# B&R Automation Studio project MotionTestBenchMaster (part 49)

```iecst
                               VAR_DOS_SEQ.Device.LTJ203.ALR_HighLimitEn := TRUE;                                      (* STEP: 9 Hema Tank Level*)
                               VAR_DOS_SEQ.Device.LTJ203.ALR_HighLimitSP := HMI_PAM_3._607;
                               VAR_DOS_SEQ.Device.LTJ203.ALR_LowLimitEn := FALSE;
                               VAR_DOS_SEQ.Device.LTJ203.ALR_LowLimitSP := 0;
                               VAR_DOS_SEQ.Device.LTJ203.SP := 55;
                               VAR_DOS_SEQ.Device.LTJ203.CMP := 3;
                               VAR_DOS_SEQ.Device.LTJ203.MinDev := 0;
                               VAR_DOS_SEQ.Device.LTJ203.MaxDev := 0;

                               VAR_DOS_SEQ.Device.TTJ203.ALR_HighLimitEn := TRUE;                                      (* STEP: 9 Hema Tank Temperature*)
                               VAR_DOS_SEQ.Device.TTJ203.ALR_HighLimitSP := HMI_PAM_3._604;
                               VAR_DOS_SEQ.Device.TTJ203.ALR_LowLimitEn := FALSE;
                               VAR_DOS_SEQ.Device.TTJ203.ALR_LowLimitSP := 0;
                               VAR_DOS_SEQ.Device.TTJ203.SP := 40;
                               VAR_DOS_SEQ.Device.TTJ203.CMP := 2;
                               VAR_DOS_SEQ.Device.TTJ203.MinDev := 0;
                               VAR_DOS_SEQ.Device.TTJ203.MaxDev := 0;

                               VAR_DOS_SEQ.Device.LSJ200.ALR := FALSE;                                                 (* STEP: 9 *)
                               VAR_DOS_SEQ.Device.LSJ200.WAIT_OFF := FALSE;
                               VAR_DOS_SEQ.Device.LSJ200.WAIT_ON := FALSE;

                               VAR_DOS_SEQ.Device.LSJ201.ALR := FALSE;                                                 (* STEP: 9 *)
                               VAR_DOS_SEQ.Device.LSJ201.WAIT_OFF := FALSE;
                               VAR_DOS_SEQ.Device.LSJ201.WAIT_ON := FALSE;

                               VAR_DOS_SEQ.Device.LSJ202.ALR := FALSE;                                                 (* STEP: 9 *)
                               VAR_DOS_SEQ.Device.LSJ202.WAIT_OFF := FALSE;
                               VAR_DOS_SEQ.Device.LSJ202.WAIT_ON := FALSE;

                               VAR_DOS_SEQ.Device.FSJ201.ALR := FALSE;                                                 (* STEP: 9 *)
                               VAR_DOS_SEQ.Device.FSJ201.WAIT_OFF := FALSE;
                               VAR_DOS_SEQ.Device.FSJ201.WAIT_ON := FALSE;

                               VAR_DOS_SEQ.Device.FSJ202.ALR := FALSE;                                                 (* STEP: 9 *)
                               VAR_DOS_SEQ.Device.FSJ202.WAIT_OFF := FALSE;
                               VAR_DOS_SEQ.Device.FSJ202.WAIT_ON := FALSE;

                               VAR_DOS_SEQ.Mem.PBAbortEnable := TRUE;                                                  (* STEP: 9 PB Abort Sequence Enable*)
                               VAR_DOS_SEQ.Mem.PBStopEnable := TRUE;                                                   (* STEP: 9 PB Stop Sequence Enable*)
                               VAR_DOS_SEQ.Mem.PBStartEnable := FALSE;                                                 (* STEP: 9 PB Start Sequence Enable*)
                               VAR_DOS_SEQ.Mem.ContainersStop := TRUE;                                                 (* STEP: 9 *)
                               VAR_DOS_SEQ.Mem.MachineStart := FALSE;                                                  (* STEP: 9 *)
                               VAR_DOS_SEQ.Mem.MachineStop := FALSE;                                                   (* STEP: 9 *)
                               VAR_DOS_SEQ.Mem.DummyBottles := FALSE;                                                  (* STEP: 9 Dummy Bottle Install*)
                               VAR_DOS_SEQ.Mem.PositioningRequest := FALSE;                                            (* STEP: 9 Request of Cam Positioning at height SP of Sequncer*)
                               VAR_DOS_SEQ.Mem.COP_Cycle := FALSE;                                                     (* STEP: 9 COP Cycle Check Requested*)
                               VAR_DOS_SEQ.Mem.LapsCounter := FALSE;                                                   (* STEP: 9 *)
                               VAR_DOS_SEQ.Mem.ValveOpening := TRUE;                                                   (* STEP: 9 *)
                               VAR_DOS_SEQ.Mem.CopAfterCipRequest := FALSE;                                            (* STEP: 9 Request Of Cop After Cip*)

                               VAR_DOS_SEQ.ITC.CIP_CleaningRequest := FALSE;                                           (* STEP: 9 To CIP -> Request of Solution Sending*)
                               VAR_DOS_SEQ.ITC.CIP_Alarm := FALSE;                                                     (* STEP: 9 To CIP -> Critical Alarm Present*)
                               VAR_DOS_SEQ.ITC.CIP_RinseEnded := FALSE;                                                (* STEP: 9 To CIP -> Rinse Finished*)
                               VAR_DOS_SEQ.ITC.CIP_ChangeEnded := FALSE;                                               (* STEP: 9 To CIP -> Change Finished*)
                               VAR_DOS_SEQ.ITC.CIP_DrainRunning := FALSE;                                              (* STEP: 9 To CIP -> Drain Cycle Running*)
                               VAR_DOS_SEQ.ITC.CIP_RinseRunning := FALSE;                                              (* STEP: 9 To CIP -> Rinse Cycle Running*)
                               VAR_DOS_SEQ.ITC.CIP_CleaningRunning := FALSE;                                           (* STEP: 9 To CIP -> Cleaning Cycle Running*)
                               VAR_DOS_SEQ.ITC.CIP_DrainEnded := FALSE;                                                (* STEP: 9 To CIP -> Drain Finished*)
                               VAR_DOS_SEQ.ITC.CIP_FloodingEnded := FALSE;                                             (* STEP: 9 To CIP -> Flooding Finished*)
                               VAR_DOS_SEQ.ITC.CIP_FlipEnable := FALSE;                                                (* STEP: 9 *)
                               VAR_DOS_SEQ.ITC.CIP_CycleEnded := FALSE;                                                (* STEP: 9 *)

                               VAR_DOS_SEQ.ITC.PROD_ReadyForHeating := TRUE;                                           (* STEP: 9 To PASTO -> Filler Ready for Production (Heating)*)
                               VAR_DOS_SEQ.ITC.PROD_DoserInTemperature := FALSE;                                       (* STEP: 9 To PASTO -> Filler Temperature OK (After Heating)*)
                               VAR_DOS_SEQ.ITC.PROD_ProductRequest := FALSE;                                           (* STEP: 9 To PASTO -> Product Request*)
                               VAR_DOS_SEQ.ITC.PROD_DoserOnFillingMode := FALSE;                                       (* STEP: 9 To PASTO -> Product Consumend -Filling Valve Opening*)
                               VAR_DOS_SEQ.ITC.PROD_EndProductionCompleted := FALSE;                                   (* STEP: 9 To PASTO -> End Production Done*)
                               VAR_DOS_SEQ.ITC.PROD_ProductRecoveryEnd := FALSE;                                       (* STEP: 9 To PASTO -> Product Recovery End*)
                               VAR_DOS_SEQ.ITC.PROD_WaterRequestAfterProd := FALSE;                                    (* STEP: 9 To PASTO -> Water Request For Filler Rinse Afetr Production*)

                       10..14: (* Spare Steps *)

                       15: (* START-UP PRODUCTION -Machine Pipes Drainages *)

                               VAR_DOS_SEQ.Device.PPJ201_PID.PID_Enable := FALSE;                                      (* STEP: 15 Doser Recovery Pump*)
                               VAR_DOS_SEQ.Device.PPJ201_PID.PID_Mode := FALSE;
                               VAR_DOS_SEQ.Device.PPJ201_PID.Auto_SP_Value := 0;
                               VAR_DOS_SEQ.Device.PPJ201_PID.FIX_Value := 0;

                               VAR_DOS_SEQ.Device.PPJ202_PID.PID_Enable := FALSE;                                      (* STEP: 15 Doser Recovery Pump*)
                               VAR_DOS_SEQ.Device.PPJ202_PID.PID_Mode := FALSE;
                               VAR_DOS_SEQ.Device.PPJ202_PID.Auto_SP_Value := 0;
                               VAR_DOS_SEQ.Device.PPJ202_PID.FIX_Value := 0;

                               VAR_DOS_SEQ.Device.PPJ203_PID.PID_Enable := FALSE;                                      (* STEP: 15 Diaphragm Pump for Recovery pulp*)
                               VAR_DOS_SEQ.Device.PPJ203_PID.PID_Mode := FALSE;
                               VAR_DOS_SEQ.Device.PPJ203_PID.Auto_SP_Value := 0;
                               VAR_DOS_SEQ.Device.PPJ203_PID.FIX_Value := 0;

                               VAR_DOS_SEQ.Device.MMJ201_PID.PID_Enable := FALSE;                                      (* STEP: 15 Shaker Motor*)
                               VAR_DOS_SEQ.Device.MMJ201_PID.PID_Mode := FALSE;
                               VAR_DOS_SEQ.Device.MMJ201_PID.Auto_SP_Value := 0;
                               VAR_DOS_SEQ.Device.MMJ201_PID.FIX_Value := 0;

                               VAR_DOS_SEQ.Device.RVJ201_PID.PID_Enable := FALSE;                                      (* STEP: 15 *)
                               VAR_DOS_SEQ.Device.RVJ201_PID.PID_Mode := FALSE;
                               VAR_DOS_SEQ.Device.RVJ201_PID.Auto_SP_Value := 0;
                               VAR_DOS_SEQ.Device.RVJ201_PID.FIX_Value := 0;

                               VAR_DOS_SEQ.Device.AVJ201.AutoCnd := FALSE;                                             (* STEP: 15 Inlet Valve*)
                               VAR_DOS_SEQ.Device.AVJ201.EnableCnd := FALSE;
                               VAR_DOS_SEQ.Device.AVJ210.AutoCnd := FALSE;                                             (* STEP: 15 Washing Duct Valve*)
                               VAR_DOS_SEQ.Device.AVJ210.EnableCnd := FALSE;
                               VAR_DOS_SEQ.Device.AVJ211.AutoCnd := FALSE;                                             (* STEP: 15 Sprayball Valve*)
                               VAR_DOS_SEQ.Device.AVJ211.EnableCnd := FALSE;
                               VAR_DOS_SEQ.Device.AVJ212.AutoCnd := FALSE;                                             (* STEP: 15 *)
                               VAR_DOS_SEQ.Device.AVJ212.EnableCnd := FALSE;
                               VAR_DOS_SEQ.Device.AVJ215.AutoCnd := TRUE;                                              (* STEP: 15 Atmospheric drain valve*)
                               VAR_DOS_SEQ.Device.AVJ215.EnableCnd := FALSE;
                               VAR_DOS_SEQ.Device.AVJ216.AutoCnd := FALSE;                                             (* STEP: 15 Recirculation Valve*)
                               VAR_DOS_SEQ.Device.AVJ216.EnableCnd := FALSE;
                               VAR_DOS_SEQ.Device.AVJ217.AutoCnd := TRUE;                                              (* STEP: 15 Tank Hema Drain Valve*)
                               VAR_DOS_SEQ.Device.AVJ217.EnableCnd := FALSE;
                               VAR_DOS_SEQ.Device.AVJ218.AutoCnd := FALSE;                                             (* STEP: 15 Recirculation Valve*)
                               VAR_DOS_SEQ.Device.AVJ218.EnableCnd := FALSE;
                               VAR_DOS_SEQ.Device.AVJ221.AutoCnd := FALSE;                                             (* STEP: 15 Inlet Loop Valve*)
                               VAR_DOS_SEQ.Device.AVJ221.EnableCnd := FALSE;
                               VAR_DOS_SEQ.Device.AVJ230.AutoCnd := FALSE;                                             (* STEP: 15 *)
                               VAR_DOS_SEQ.Device.AVJ230.EnableCnd := FALSE;
                               VAR_DOS_SEQ.Device.AVJ231.AutoCnd := FALSE;                                             (* STEP: 15 *)
                               VAR_DOS_SEQ.Device.AVJ231.EnableCnd := FALSE;
                               VAR_DOS_SEQ.Device.AVJ232.AutoCnd := TRUE;                                              (* STEP: 15 *)
                               VAR_DOS_SEQ.Device.AVJ232.EnableCnd := FALSE;
                               VAR_DOS_SEQ.Device.AVJ233.AutoCnd := FALSE;                                             (* STEP: 15 *)
                               VAR_DOS_SEQ.Device.AVJ233.EnableCnd := FALSE;
                               VAR_DOS_SEQ.Device.AVJ234.AutoCnd := FALSE;                                             (* STEP: 15 *)
                               VAR_DOS_SEQ.Device.AVJ234.EnableCnd := FALSE;
                               VAR_DOS_SEQ.Device.AVJ235.AutoCnd := TRUE;                                              (* STEP: 15 *)
                               VAR_DOS_SEQ.Device.AVJ235.EnableCnd := FALSE;

                               VAR_DOS_SEQ.Device.LTJ203.ALR_HighLimitEn := FALSE;                                     (* STEP: 15 Hema Tank Level*)
                               VAR_DOS_SEQ.Device.LTJ203.ALR_HighLimitSP := 0;
                               VAR_DOS_SEQ.Device.LTJ203.ALR_LowLimitEn := FALSE;
                               VAR_DOS_SEQ.Device.LTJ203.ALR_LowLimitSP := 0;
                               VAR_DOS_SEQ.Device.LTJ203.SP := 5;
                               VAR_DOS_SEQ.Device.LTJ203.CMP := 1;
                               VAR_DOS_SEQ.Device.LTJ203.MinDev := 1;
                               VAR_DOS_SEQ.Device.LTJ203.MaxDev := 1;

                               VAR_DOS_SEQ.Device.TTJ203.ALR_HighLimitEn := FALSE;                                     (* STEP: 15 Hema Tank Temperature*)
                               VAR_DOS_SEQ.Device.TTJ203.ALR_HighLimitSP := 0;
                               VAR_DOS_SEQ.Device.TTJ203.ALR_LowLimitEn := FALSE;
                               VAR_DOS_SEQ.Device.TTJ203.ALR_LowLimitSP := 0;
                               VAR_DOS_SEQ.Device.TTJ203.SP := 0;
                               VAR_DOS_SEQ.Device.TTJ203.CMP := 0;
                               VAR_DOS_SEQ.Device.TTJ203.MinDev := 0;
                               VAR_DOS_SEQ.Device.TTJ203.MaxDev := 0;

                               VAR_DOS_SEQ.Device.LSJ200.ALR := FALSE;                                                 (* STEP: 15 *)
                               VAR_DOS_SEQ.Device.LSJ200.WAIT_OFF := FALSE;
                               VAR_DOS_SEQ.Device.LSJ200.WAIT_ON := FALSE;

                               VAR_DOS_SEQ.Device.LSJ201.ALR := FALSE;                                                 (* STEP: 15 *)
                               VAR_DOS_SEQ.Device.LSJ201.WAIT_OFF := FALSE;
                               VAR_DOS_SEQ.Device.LSJ201.WAIT_ON := FALSE;

                               VAR_DOS_SEQ.Device.LSJ202.ALR := FALSE;                                                 (* STEP: 15 *)
                               VAR_DOS_SEQ.Device.LSJ202.WAIT_OFF := FALSE;
                               VAR_DOS_SEQ.Device.LSJ202.WAIT_ON := FALSE;

                               VAR_DOS_SEQ.Device.FSJ201.ALR := FALSE;                                                 (* STEP: 15 *)
                               VAR_DOS_SEQ.Device.FSJ201.WAIT_OFF := FALSE;
                               VAR_DOS_SEQ.Device.FSJ201.WAIT_ON := FALSE;

                               VAR_DOS_SEQ.Device.FSJ202.ALR := FALSE;                                                 (* STEP: 15 *)
                               VAR_DOS_SEQ.Device.FSJ202.WAIT_OFF := FALSE;
                               VAR_DOS_SEQ.Device.FSJ202.WAIT_ON := FALSE;

                               VAR_DOS_SEQ.Mem.PBAbortEnable := TRUE;                                                  (* STEP: 15 PB Abort Sequence Enable*)
                               VAR_DOS_SEQ.Mem.PBStopEnable := TRUE;                                                   (* STEP: 15 PB Stop Sequence Enable*)
                               VAR_DOS_SEQ.Mem.PBStartEnable := FALSE;                                                 (* STEP: 15 PB Start Sequence Enable*)
                               VAR_DOS_SEQ.Mem.ContainersStop := TRUE;                                                (* STEP: 15 *)
                               VAR_DOS_SEQ.Mem.MachineStart := TRUE;                                                   (* STEP: 15 *)
                               VAR_DOS_SEQ.Mem.MachineStop := FALSE;                                                   (* STEP: 15 *)
                               VAR_DOS_SEQ.Mem.DummyBottles := FALSE;                                                  (* STEP: 15 Dummy Bottle Install*)
                               VAR_DOS_SEQ.Mem.PositioningRequest := FALSE;                                            (* STEP: 15 Request of Cam Positioning at height SP of Sequncer*)
                               VAR_DOS_SEQ.Mem.COP_Cycle := FALSE;                                                     (* STEP: 15 COP Cycle Check Requested*)
                               VAR_DOS_SEQ.Mem.LapsCounter := FALSE;                                                   (* STEP: 15 *)
                               VAR_DOS_SEQ.Mem.ValveOpening := FALSE;                                                  (* STEP: 15 *)
                               VAR_DOS_SEQ.Mem.CopAfterCipRequest := FALSE;                                            (* STEP: 15 Request Of Cop After Cip*)

                               VAR_DOS_SEQ.ITC.CIP_CleaningRequest := FALSE;                                           (* STEP: 15 To CIP -> Request of Solution Sending*)
                               VAR_DOS_SEQ.ITC.CIP_Alarm := FALSE;                                                     (* STEP: 15 To CIP -> Critical Alarm Present*)
                               VAR_DOS_SEQ.ITC.CIP_RinseEnded := FALSE;                                                (* STEP: 15 To CIP -> Rinse Finished*)
                               VAR_DOS_SEQ.ITC.CIP_ChangeEnded := FALSE;                                               (* STEP: 15 To CIP -> Change Finished*)
                               VAR_DOS_SEQ.ITC.CIP_DrainRunning := FALSE;                                              (* STEP: 15 To CIP -> Drain Cycle Running*)
                               VAR_DOS_SEQ.ITC.CIP_RinseRunning := FALSE;                                              (* STEP: 15 To CIP -> Rinse Cycle Running*)
                               VAR_DOS_SEQ.ITC.CIP_CleaningRunning := FALSE;                                           (* STEP: 15 To CIP -> Cleaning Cycle Running*)
                               VAR_DOS_SEQ.ITC.CIP_DrainEnded := FALSE;                                                (* STEP: 15 To CIP -> Drain Finished*)
                               VAR_DOS_SEQ.ITC.CIP_FloodingEnded := FALSE;                                             (* STEP: 15 To CIP -> Flooding Finished*)
                               VAR_DOS_SEQ.ITC.CIP_FlipEnable := FALSE;                                                (* STEP: 15 *)
                               VAR_DOS_SEQ.ITC.CIP_CycleEnded := FALSE;                                                (* STEP: 15 *)

                               VAR_DOS_SEQ.ITC.PROD_ReadyForHeating := FALSE;                                          (* STEP: 15 To PASTO -> Filler Ready for Production (Heating)*)
                               VAR_DOS_SEQ.ITC.PROD_DoserInTemperature := TRUE;                                        (* STEP: 15 To PASTO -> Filler Temperature OK (After Heating)*)
                               VAR_DOS_SEQ.ITC.PROD_ProductRequest := FALSE;                                           (* STEP: 15 To PASTO -> Product Request*)
                               VAR_DOS_SEQ.ITC.PROD_DoserOnFillingMode := FALSE;                                       (* STEP: 15 To PASTO -> Product Consumend -Filling Valve Opening*)
                               VAR_DOS_SEQ.ITC.PROD_EndProductionCompleted := FALSE;                                   (* STEP: 15 To PASTO -> End Production Done*)
                               VAR_DOS_SEQ.ITC.PROD_ProductRecoveryEnd := FALSE;                                       (* STEP: 15 To PASTO -> Product Recovery End*)
                               VAR_DOS_SEQ.ITC.PROD_WaterRequestAfterProd := FALSE;                                    (* STEP: 15 To PASTO -> Water Request For Filler Rinse Afetr Production*)

                       16: (* Spare Steps *)

                       17: (* START-UP PRODUCTION -Machine Draining End *)

                               VAR_DOS_SEQ.Device.PPJ201_PID.PID_Enable := FALSE;                                      (* STEP: 17 Doser Recovery Pump*)
                               VAR_DOS_SEQ.Device.PPJ201_PID.PID_Mode := FALSE;
                               VAR_DOS_SEQ.Device.PPJ201_PID.Auto_SP_Value := 0;
                               VAR_DOS_SEQ.Device.PPJ201_PID.FIX_Value := 0;

                               VAR_DOS_SEQ.Device.PPJ202_PID.PID_Enable := FALSE;                                      (* STEP: 17 Doser Recovery Pump*)
                               VAR_DOS_SEQ.Device.PPJ202_PID.PID_Mode := FALSE;
                               VAR_DOS_SEQ.Device.PPJ202_PID.Auto_SP_Value := 0;
                               VAR_DOS_SEQ.Device.PPJ202_PID.FIX_Value := 0;

                               VAR_DOS_SEQ.Device.PPJ203_PID.PID_Enable := FALSE;                                      (* STEP: 17 Diaphragm Pump for Recovery pulp*)
                               VAR_DOS_SEQ.Device.PPJ203_PID.PID_Mode := FALSE;
                               VAR_DOS_SEQ.Device.PPJ203_PID.Auto_SP_Value := 0;
                               VAR_DOS_SEQ.Device.PPJ203_PID.FIX_Value := 0;

                               VAR_DOS_SEQ.Device.MMJ201_PID.PID_Enable := FALSE;                                      (* STEP: 17 Shaker Motor*)
                               VAR_DOS_SEQ.Device.MMJ201_PID.PID_Mode := FALSE;
                               VAR_DOS_SEQ.Device.MMJ201_PID.Auto_SP_Value := 0;
                               VAR_DOS_SEQ.Device.MMJ201_PID.FIX_Value := 0;

                               VAR_DOS_SEQ.Device.RVJ201_PID.PID_Enable := FALSE;                                      (* STEP: 17 *)
                               VAR_DOS_SEQ.Device.RVJ201_PID.PID_Mode := FALSE;
                               VAR_DOS_SEQ.Device.RVJ201_PID.Auto_SP_Value := 0;
                               VAR_DOS_SEQ.Device.RVJ201_PID.FIX_Value := 0;

                               VAR_DOS_SEQ.Device.AVJ201.AutoCnd := FALSE;                                             (* STEP: 17 Inlet Valve*)
                               VAR_DOS_SEQ.Device.AVJ201.EnableCnd := FALSE;
                               VAR_DOS_SEQ.Device.AVJ210.AutoCnd := FALSE;                                             (* STEP: 17 Washing Duct Valve*)
                               VAR_DOS_SEQ.Device.AVJ210.EnableCnd := FALSE;
                               VAR_DOS_SEQ.Device.AVJ211.AutoCnd := FALSE;                                             (* STEP: 17 Sprayball Valve*)
                               VAR_DOS_SEQ.Device.AVJ211.EnableCnd := FALSE;
                               VAR_DOS_SEQ.Device.AVJ212.AutoCnd := FALSE;                                             (* STEP: 17 *)
                               VAR_DOS_SEQ.Device.AVJ212.EnableCnd := FALSE;
                               VAR_DOS_SEQ.Device.AVJ215.AutoCnd := TRUE;                                              (* STEP: 17 Atmospheric drain valve*)
                               VAR_DOS_SEQ.Device.AVJ215.EnableCnd := FALSE;
                               VAR_DOS_SEQ.Device.AVJ216.AutoCnd := FALSE;                                             (* STEP: 17 Recirculation Valve*)
                               VAR_DOS_SEQ.Device.AVJ216.EnableCnd := FALSE;
                               VAR_DOS_SEQ.Device.AVJ217.AutoCnd := TRUE;                                              (* STEP: 17 Tank Hema Drain Valve*)
                               VAR_DOS_SEQ.Device.AVJ217.EnableCnd := FALSE;
                               VAR_DOS_SEQ.Device.AVJ218.AutoCnd := FALSE;                                             (* STEP: 17 Recirculation Valve*)
                               VAR_DOS_SEQ.Device.AVJ218.EnableCnd := FALSE;
                               VAR_DOS_SEQ.Device.AVJ221.AutoCnd := FALSE;                                             (* STEP: 17 Inlet Loop Valve*)
                               VAR_DOS_SEQ.Device.AVJ221.EnableCnd := FALSE;
                               VAR_DOS_SEQ.Device.AVJ230.AutoCnd := FALSE;                                             (* STEP: 17 *)
                               VAR_DOS_SEQ.Device.AVJ230.EnableCnd := FALSE;
                               VAR_DOS_SEQ.Device.AVJ231.AutoCnd := FALSE;                                             (* STEP: 17 *)
                               VAR_DOS_SEQ.Device.AVJ231.EnableCnd := FALSE;
                               VAR_DOS_SEQ.Device.AVJ232.AutoCnd := TRUE;                                              (* STEP: 17 *)
                               VAR_DOS_SEQ.Device.AVJ232.EnableCnd := FALSE;
                               VAR_DOS_SEQ.Device.AVJ233.AutoCnd := FALSE;                                             (* STEP: 17 *)
                               VAR_DOS_SEQ.Device.AVJ233.EnableCnd := FALSE;
                               VAR_DOS_SEQ.Device.AVJ234.AutoCnd := FALSE;                                             (* STEP: 17 *)
                               VAR_DOS_SEQ.Device.AVJ234.EnableCnd := FALSE;
                               VAR_DOS_SEQ.Device.AVJ235.AutoCnd := TRUE;                                              (* STEP: 17 *)
                               VAR_DOS_SEQ.Device.AVJ235.EnableCnd := FALSE;

                               VAR_DOS_SEQ.Device.LTJ203.ALR_HighLimitEn := FALSE;                                     (* STEP: 17 Hema Tank Level*)
                               VAR_DOS_SEQ.Device.LTJ203.ALR_HighLimitSP := 0;
                               VAR_DOS_SEQ.Device.LTJ203.ALR_LowLimitEn := FALSE;
                               VAR_DOS_SEQ.Device.LTJ203.ALR_LowLimitSP := 0;
                               VAR_DOS_SEQ.Device.LTJ203.SP := 0;
                               VAR_DOS_SEQ.Device.LTJ203.CMP := 0;
                               VAR_DOS_SEQ.Device.LTJ203.MinDev := 0;
                               VAR_DOS_SEQ.Device.LTJ203.MaxDev := 0;

                               VAR_DOS_SEQ.Device.TTJ203.ALR_HighLimitEn := FALSE;                                     (* STEP: 17 Hema Tank Temperature*)
                               VAR_DOS_SEQ.Device.TTJ203.ALR_HighLimitSP := 0;
                               VAR_DOS_SEQ.Device.TTJ203.ALR_LowLimitEn := FALSE;
                               VAR_DOS_SEQ.Device.TTJ203.ALR_LowLimitSP := 0;
                               VAR_DOS_SEQ.Device.TTJ203.SP := 0;
                               VAR_DOS_SEQ.Device.TTJ203.CMP := 0;
                               VAR_DOS_SEQ.Device.TTJ203.MinDev := 0;
                               VAR_DOS_SEQ.Device.TTJ203.MaxDev := 0;

                               VAR_DOS_SEQ.Device.LSJ200.ALR := FALSE;                                                 (* STEP: 17 *)
                               VAR_DOS_SEQ.Device.LSJ200.WAIT_OFF := FALSE;
                               VAR_DOS_SEQ.Device.LSJ200.WAIT_ON := FALSE;

                               VAR_DOS_SEQ.Device.LSJ201.ALR := FALSE;                                                 (* STEP: 17 *)
                               VAR_DOS_SEQ.Device.LSJ201.WAIT_OFF := FALSE;
                               VAR_DOS_SEQ.Device.LSJ201.WAIT_ON := FALSE;

                               VAR_DOS_SEQ.Device.LSJ202.ALR := FALSE;                                                 (* STEP: 17 *)
                               VAR_DOS_SEQ.Device.LSJ202.WAIT_OFF := FALSE;
                               VAR_DOS_SEQ.Device.LSJ202.WAIT_ON := FALSE;

                               VAR_DOS_SEQ.Device.FSJ201.ALR := FALSE;                                                 (* STEP: 17 *)
                               VAR_DOS_SEQ.Device.FSJ201.WAIT_OFF := FALSE;
                               VAR_DOS_SEQ.Device.FSJ201.WAIT_ON := FALSE;

                               VAR_DOS_SEQ.Device.FSJ202.ALR := FALSE;                                                 (* STEP: 17 *)
                               VAR_DOS_SEQ.Device.FSJ202.WAIT_OFF := FALSE;
                               VAR_DOS_SEQ.Device.FSJ202.WAIT_ON := FALSE;

                               VAR_DOS_SEQ.Mem.PBAbortEnable := TRUE;                                                  (* STEP: 17 PB Abort Sequence Enable*)
                               VAR_DOS_SEQ.Mem.PBStopEnable := TRUE;                                                   (* STEP: 17 PB Stop Sequence Enable*)
                               VAR_DOS_SEQ.Mem.PBStartEnable := FALSE;                                                 (* STEP: 17 PB Start Sequence Enable*)
                               VAR_DOS_SEQ.Mem.ContainersStop := TRUE;                                                 (* STEP: 17 *)
                               VAR_DOS_SEQ.Mem.MachineStart := FALSE;                                                  (* STEP: 17 *)
                               VAR_DOS_SEQ.Mem.MachineStop := FALSE;                                                   (* STEP: 17 *)
                               VAR_DOS_SEQ.Mem.DummyBottles := FALSE;                                                  (* STEP: 17 Dummy Bottle Install*)
                               VAR_DOS_SEQ.Mem.PositioningRequest := FALSE;                                            (* STEP: 17 Request of Cam Positioning at height SP of Sequncer*)
                               VAR_DOS_SEQ.Mem.COP_Cycle := FALSE;                                                     (* STEP: 17 COP Cycle Check Requested*)
                               VAR_DOS_SEQ.Mem.LapsCounter := FALSE;                                                   (* STEP: 17 *)
                               VAR_DOS_SEQ.Mem.ValveOpening := FALSE;                                                  (* STEP: 17 *)
                               VAR_DOS_SEQ.Mem.CopAfterCipRequest := FALSE;                                            (* STEP: 17 Request Of Cop After Cip*)

                               VAR_DOS_SEQ.ITC.CIP_CleaningRequest := FALSE;                                           (* STEP: 17 To CIP -> Request of Solution Sending*)
                               VAR_DOS_SEQ.ITC.CIP_Alarm := FALSE;                                                     (* STEP: 17 To CIP -> Critical Alarm Present*)
                               VAR_DOS_SEQ.ITC.CIP_RinseEnded := FALSE;                                                (* STEP: 17 To CIP -> Rinse Finished*)
                               VAR_DOS_SEQ.ITC.CIP_ChangeEnded := FALSE;                                               (* STEP: 17 To CIP -> Change Finished*)
                               VAR_DOS_SEQ.ITC.CIP_DrainRunning := FALSE;                                              (* STEP: 17 To CIP -> Drain Cycle Running*)
                               VAR_DOS_SEQ.ITC.CIP_RinseRunning := FALSE;                                              (* STEP: 17 To CIP -> Rinse Cycle Running*)
                               VAR_DOS_SEQ.ITC.CIP_CleaningRunning := FALSE;                                           (* STEP: 17 To CIP -> Cleaning Cycle Running*)
                               VAR_DOS_SEQ.ITC.CIP_DrainEnded := FALSE;                                                (* STEP: 17 To CIP -> Drain Finished*)
                               VAR_DOS_SEQ.ITC.CIP_FloodingEnded := FALSE;                                             (* STEP: 17 To CIP -> Flooding Finished*)
                               VAR_DOS_SEQ.ITC.CIP_FlipEnable := FALSE;                                                (* STEP: 17 *)
                               VAR_DOS_SEQ.ITC.CIP_CycleEnded := FALSE;                                                (* STEP: 17 *)

                               VAR_DOS_SEQ.ITC.PROD_ReadyForHeating := FALSE;                                          (* STEP: 17 To PASTO -> Filler Ready for Production (Heating)*)
                               VAR_DOS_SEQ.ITC.PROD_DoserInTemperature := FALSE;                                       (* STEP: 17 To PASTO -> Filler Temperature OK (After Heating)*)
                               VAR_DOS_SEQ.ITC.PROD_ProductRequest := FALSE;                                           (* STEP: 17 To PASTO -> Product Request*)
                               VAR_DOS_SEQ.ITC.PROD_DoserOnFillingMode := FALSE;                                       (* STEP: 17 To PASTO -> Product Consumend -Filling Valve Opening*)
                               VAR_DOS_SEQ.ITC.PROD_EndProductionCompleted := FALSE;                                   (* STEP: 17 To PASTO -> End Production Done*)
                               VAR_DOS_SEQ.ITC.PROD_ProductRecoveryEnd := FALSE;                                       (* STEP: 17 To PASTO -> Product Recovery End*)
                               VAR_DOS_SEQ.ITC.PROD_WaterRequestAfterProd := FALSE;                                    (* STEP: 17 To PASTO -> Water Request For Filler Rinse Afetr Production*)

                       18..19: (* Spare Steps *)

                       20: (* START-UP PRODUCTION -Wait "Product Available" From PASTO *)

                               VAR_DOS_SEQ.Device.PPJ201_PID.PID_Enable := FALSE;                                      (* STEP: 20 Doser Recovery Pump*)
                               VAR_DOS_SEQ.Device.PPJ201_PID.PID_Mode := FALSE;
                               VAR_DOS_SEQ.Device.PPJ201_PID.Auto_SP_Value := 0;
                               VAR_DOS_SEQ.Device.PPJ201_PID.FIX_Value := 0;

                               VAR_DOS_SEQ.Device.PPJ202_PID.PID_Enable := FALSE;                                      (* STEP: 20 Doser Recovery Pump*)
                               VAR_DOS_SEQ.Device.PPJ202_PID.PID_Mode := FALSE;
                               VAR_DOS_SEQ.Device.PPJ202_PID.Auto_SP_Value := 0;
                               VAR_DOS_SEQ.Device.PPJ202_PID.FIX_Value := 0;

                               VAR_DOS_SEQ.Device.PPJ203_PID.PID_Enable := FALSE;                                      (* STEP: 20 Diaphragm Pump for Recovery pulp*)
                               VAR_DOS_SEQ.Device.PPJ203_PID.PID_Mode := FALSE;
                               VAR_DOS_SEQ.Device.PPJ203_PID.Auto_SP_Value := 0;
                               VAR_DOS_SEQ.Device.PPJ203_PID.FIX_Value := 0;

                               VAR_DOS_SEQ.Device.MMJ201_PID.PID_Enable := FALSE;                                      (* STEP: 20 Shaker Motor*)
                               VAR_DOS_SEQ.Device.MMJ201_PID.PID_Mode := FALSE;
                               VAR_DOS_SEQ.Device.MMJ201_PID.Auto_SP_Value := 0;
                               VAR_DOS_SEQ.Device.MMJ201_PID.FIX_Value := 0;

                               VAR_DOS_SEQ.Device.RVJ201_PID.PID_Enable := FALSE;                                      (* STEP: 20 *)
                               VAR_DOS_SEQ.Device.RVJ201_PID.PID_Mode := FALSE;
                               VAR_DOS_SEQ.Device.RVJ201_PID.Auto_SP_Value := 0;
                               VAR_DOS_SEQ.Device.RVJ201_PID.FIX_Value := 0;

                               VAR_DOS_SEQ.Device.AVJ201.AutoCnd := FALSE;                                             (* STEP: 20 Inlet Valve*)
                               VAR_DOS_SEQ.Device.AVJ201.EnableCnd := FALSE;
                               VAR_DOS_SEQ.Device.AVJ210.AutoCnd := FALSE;                                             (* STEP: 20 Washing Duct Valve*)
                               VAR_DOS_SEQ.Device.AVJ210.EnableCnd := FALSE;
                               VAR_DOS_SEQ.Device.AVJ211.AutoCnd := FALSE;                                             (* STEP: 20 Sprayball Valve*)
                               VAR_DOS_SEQ.Device.AVJ211.EnableCnd := FALSE;
                               VAR_DOS_SEQ.Device.AVJ212.AutoCnd := FALSE;                                             (* STEP: 20 *)
                               VAR_DOS_SEQ.Device.AVJ212.EnableCnd := FALSE;
                               VAR_DOS_SEQ.Device.AVJ215.AutoCnd := TRUE;                                              (* STEP: 20 Atmospheric drain valve *)
                               VAR_DOS_SEQ.Device.AVJ215.EnableCnd := FALSE;
                               VAR_DOS_SEQ.Device.AVJ216.AutoCnd := FALSE;                                             (* STEP: 20 Recirculation Valve*)
                               VAR_DOS_SEQ.Device.AVJ216.EnableCnd := FALSE;
                               VAR_DOS_SEQ.Device.AVJ217.AutoCnd := FALSE;                                              (* STEP: 20 Tank Hema Drain Valve*)
                               VAR_DOS_SEQ.Device.AVJ217.EnableCnd := FALSE;
                               VAR_DOS_SEQ.Device.AVJ218.AutoCnd := FALSE;                                             (* STEP: 20 Recirculation Valve*)
                               VAR_DOS_SEQ.Device.AVJ218.EnableCnd := FALSE;
                               VAR_DOS_SEQ.Device.AVJ221.AutoCnd := FALSE;                                             (* STEP: 20 Inlet Loop Valve*)
                               VAR_DOS_SEQ.Device.AVJ221.EnableCnd := FALSE;
                               VAR_DOS_SEQ.Device.AVJ230.AutoCnd := FALSE;                                             (* STEP: 20 *)
                               VAR_DOS_SEQ.Device.AVJ230.EnableCnd := FALSE;
                               VAR_DOS_SEQ.Device.AVJ231.AutoCnd := FALSE;                                             (* STEP: 20 *)
                               VAR_DOS_SEQ.Device.AVJ231.EnableCnd := FALSE;
                               VAR_DOS_SEQ.Device.AVJ232.AutoCnd := FALSE;                                             (* STEP: 20 *)
                               VAR_DOS_SEQ.Device.AVJ232.EnableCnd := FALSE;
                               VAR_DOS_SEQ.Device.AVJ233.AutoCnd := FALSE;                                             (* STEP: 20 *)
                               VAR_DOS_SEQ.Device.AVJ233.EnableCnd := FALSE;
                               VAR_DOS_SEQ.Device.AVJ234.AutoCnd := FALSE;                                             (* STEP: 20 *)
                               VAR_DOS_SEQ.Device.AVJ234.EnableCnd := FALSE;
                               VAR_DOS_SEQ.Device.AVJ235.AutoCnd := FALSE;                                             (* STEP: 20 *)
                               VAR_DOS_SEQ.Device.AVJ235.EnableCnd := FALSE;

                               VAR_DOS_SEQ.Device.LTJ203.ALR_HighLimitEn := FALSE;                                     (* STEP: 20 Hema Tank Level*)
                               VAR_DOS_SEQ.Device.LTJ203.ALR_HighLimitSP := 0;
                               VAR_DOS_SEQ.Device.LTJ203.ALR_LowLimitEn := FALSE;
                               VAR_DOS_SEQ.Device.LTJ203.ALR_LowLimitSP := 0;
                               VAR_DOS_SEQ.Device.LTJ203.SP := 0;
                               VAR_DOS_SEQ.Device.LTJ203.CMP := 0;
                               VAR_DOS_SEQ.Device.LTJ203.MinDev := 0;
                               VAR_DOS_SEQ.Device.LTJ203.MaxDev := 0;

                               VAR_DOS_SEQ.Device.TTJ203.ALR_HighLimitEn := FALSE;                                     (* STEP: 20 Hema Tank Temperature*)
                               VAR_DOS_SEQ.Device.TTJ203.ALR_HighLimitSP := 0;
                               VAR_DOS_SEQ.Device.TTJ203.ALR_LowLimitEn := FALSE;
                               VAR_DOS_SEQ.Device.TTJ203.ALR_LowLimitSP := 0;
                               VAR_DOS_SEQ.Device.TTJ203.SP := 0;
                               VAR_DOS_SEQ.Device.TTJ203.CMP := 0;
                               VAR_DOS_SEQ.Device.TTJ203.MinDev := 0;
                               VAR_DOS_SEQ.Device.TTJ203.MaxDev := 0;

                               VAR_DOS_SEQ.Device.LSJ200.ALR := FALSE;                                                 (* STEP: 20 *)
                               VAR_DOS_SEQ.Device.LSJ200.WAIT_OFF := FALSE;
                               VAR_DOS_SEQ.Device.LSJ200.WAIT_ON := FALSE;

                               VAR_DOS_SEQ.Device.LSJ201.ALR := FALSE;                                                 (* STEP: 20 *)
                               VAR_DOS_SEQ.Device.LSJ201.WAIT_OFF := FALSE;
                               VAR_DOS_SEQ.Device.LSJ201.WAIT_ON := FALSE;

                               VAR_DOS_SEQ.Device.LSJ202.ALR := FALSE;                                                 (* STEP: 20 *)
                               VAR_DOS_SEQ.Device.LSJ202.WAIT_OFF := FALSE;
                               VAR_DOS_SEQ.Device.LSJ202.WAIT_ON := FALSE;

                               VAR_DOS_SEQ.Device.FSJ201.ALR := FALSE;                                                 (* STEP: 20 *)
                               VAR_DOS_SEQ.Device.FSJ201.WAIT_OFF := FALSE;
                               VAR_DOS_SEQ.Device.FSJ201.WAIT_ON := FALSE;

                               VAR_DOS_SEQ.Device.FSJ202.ALR := FALSE;                                                 (* STEP: 20 *)
                               VAR_DOS_SEQ.Device.FSJ202.WAIT_OFF := FALSE;
                               VAR_DOS_SEQ.Device.FSJ202.WAIT_ON := FALSE;

                               VAR_DOS_SEQ.Mem.PBAbortEnable := TRUE;                                                  (* STEP: 20 PB Abort Sequence Enable*)
                               VAR_DOS_SEQ.Mem.PBStopEnable := TRUE;                                                   (* STEP: 20 PB Stop Sequence Enable*)
                               VAR_DOS_SEQ.Mem.PBStartEnable := FALSE;                                                 (* STEP: 20 PB Start Sequence Enable*)
                               VAR_DOS_SEQ.Mem.ContainersStop := TRUE;                                                 (* STEP: 20 *)
                               VAR_DOS_SEQ.Mem.MachineStart := FALSE;                                                  (* STEP: 20 *)
                               VAR_DOS_SEQ.Mem.MachineStop := FALSE;                                                   (* STEP: 20 *)
                               VAR_DOS_SEQ.Mem.DummyBottles := FALSE;                                                  (* STEP: 20 Dummy Bottle Install*)
                               VAR_DOS_SEQ.Mem.PositioningRequest := FALSE;                                            (* STEP: 20 Request of Cam Positioning at height SP of Sequncer*)
                               VAR_DOS_SEQ.Mem.COP_Cycle := FALSE;                                                     (* STEP: 20 COP Cycle Check Requested*)
                               VAR_DOS_SEQ.Mem.LapsCounter := FALSE;                                                   (* STEP: 20 *)
                               VAR_DOS_SEQ.Mem.ValveOpening := FALSE;                                                  (* STEP: 20 *)
                               VAR_DOS_SEQ.Mem.CopAfterCipRequest := FALSE;                                            (* STEP: 20 Request Of Cop After Cip*)

                               VAR_DOS_SEQ.ITC.CIP_CleaningRequest := FALSE;                                           (* STEP: 20 To CIP -> Request of Solution Sending*)
                               VAR_DOS_SEQ.ITC.CIP_Alarm := FALSE;                                                     (* STEP: 20 To CIP -> Critical Alarm Present*)
                               VAR_DOS_SEQ.ITC.CIP_RinseEnded := FALSE;                                                (* STEP: 20 To CIP -> Rinse Finished*)
                               VAR_DOS_SEQ.ITC.CIP_ChangeEnded := FALSE;                                               (* STEP: 20 To CIP -> Change Finished*)
                               VAR_DOS_SEQ.ITC.CIP_DrainRunning := FALSE;                                              (* STEP: 20 To CIP -> Drain Cycle Running*)
                               VAR_DOS_SEQ.ITC.CIP_RinseRunning := FALSE;                                              (* STEP: 20 To CIP -> Rinse Cycle Running*)
                               VAR_DOS_SEQ.ITC.CIP_CleaningRunning := FALSE;                                           (* STEP: 20 To CIP -> Cleaning Cycle Running*)
                               VAR_DOS_SEQ.ITC.CIP_DrainEnded := FALSE;                                                (* STEP: 20 To CIP -> Drain Finished*)
                               VAR_DOS_SEQ.ITC.CIP_FloodingEnded := FALSE;                                             (* STEP: 20 To CIP -> Flooding Finished*)
                               VAR_DOS_SEQ.ITC.CIP_FlipEnable := FALSE;                                                (* STEP: 20 *)
                               VAR_DOS_SEQ.ITC.CIP_CycleEnded := FALSE;                                                (* STEP: 20 *)

                               VAR_DOS_SEQ.ITC.PROD_ReadyForHeating := FALSE;                                          (* STEP: 20 To PASTO -> Filler Ready for Production (Heating)*)
                               VAR_DOS_SEQ.ITC.PROD_DoserInTemperature := FALSE;                                       (* STEP: 20 To PASTO -> Filler Temperature OK (After Heating)*)
                               VAR_DOS_SEQ.ITC.PROD_ProductRequest := FALSE;                                           (* STEP: 20 To PASTO -> Product Request*)
                               VAR_DOS_SEQ.ITC.PROD_DoserOnFillingMode := FALSE;                                       (* STEP: 20 To PASTO -> Product Consumend -Filling Valve Opening*)
                               VAR_DOS_SEQ.ITC.PROD_EndProductionCompleted := FALSE;                                   (* STEP: 20 To PASTO -> End Production Done*)
                               VAR_DOS_SEQ.ITC.PROD_ProductRecoveryEnd := FALSE;                                       (* STEP: 20 To PASTO -> Product Recovery End*)
                               VAR_DOS_SEQ.ITC.PROD_WaterRequestAfterProd := FALSE;                                    (* STEP: 20 To PASTO -> Water Request For Filler Rinse Afetr Production*)

                       21: (* Spare Steps *)

                       22: (* START-UP PRODUCTION - Load Product at level *)

                               VAR_DOS_SEQ.Device.PPJ201_PID.PID_Enable := FALSE;                                      (* STEP: 22 Doser Recovery Pump*)
                               VAR_DOS_SEQ.Device.PPJ201_PID.PID_Mode := FALSE;
                               VAR_DOS_SEQ.Device.PPJ201_PID.Auto_SP_Value := 0;
                               VAR_DOS_SEQ.Device.PPJ201_PID.FIX_Value := 0;

                               VAR_DOS_SEQ.Device.PPJ202_PID.PID_Enable := FALSE;                                      (* STEP: 22 Doser Recovery Pump*)
                               VAR_DOS_SEQ.Device.PPJ202_PID.PID_Mode := FALSE;
                               VAR_DOS_SEQ.Device.PPJ202_PID.Auto_SP_Value := 0;
                               VAR_DOS_SEQ.Device.PPJ202_PID.FIX_Value := 0;

                               VAR_DOS_SEQ.Device.PPJ203_PID.PID_Enable := FALSE;                                      (* STEP: 22 Diaphragm Pump for Recovery pulp*)
                               VAR_DOS_SEQ.Device.PPJ203_PID.PID_Mode := FALSE;
                               VAR_DOS_SEQ.Device.PPJ203_PID.Auto_SP_Value := 0;
                               VAR_DOS_SEQ.Device.PPJ203_PID.FIX_Value := 0;

                               VAR_DOS_SEQ.Device.MMJ201_PID.PID_Enable := FALSE;                                      (* STEP: 22 Shaker Motor*)
                               VAR_DOS_SEQ.Device.MMJ201_PID.PID_Mode := FALSE;
                               VAR_DOS_SEQ.Device.MMJ201_PID.Auto_SP_Value := 10;
                               VAR_DOS_SEQ.Device.MMJ201_PID.FIX_Value := 0;

                               VAR_DOS_SEQ.Device.RVJ201_PID.PID_Enable := FALSE;                                      (* STEP: 22 *)
                               VAR_DOS_SEQ.Device.RVJ201_PID.PID_Mode := FALSE;
                               VAR_DOS_SEQ.Device.RVJ201_PID.Auto_SP_Value := 0;
                               VAR_DOS_SEQ.Device.RVJ201_PID.FIX_Value := 0;

                               VAR_DOS_SEQ.Device.AVJ201.AutoCnd := TRUE;                                              (* STEP: 22 Inlet Valve*)
                               VAR_DOS_SEQ.Device.AVJ201.EnableCnd := TRUE;
                               VAR_DOS_SEQ.Device.AVJ210.AutoCnd := FALSE;                                             (* STEP: 22 Washing Duct Valve*)
                               VAR_DOS_SEQ.Device.AVJ210.EnableCnd := FALSE;
                               VAR_DOS_SEQ.Device.AVJ211.AutoCnd := FALSE;                                             (* STEP: 22 Sprayball Valve*)
                               VAR_DOS_SEQ.Device.AVJ211.EnableCnd := FALSE;
                               VAR_DOS_SEQ.Device.AVJ212.AutoCnd := FALSE;                                             (* STEP: 22 *)
                               VAR_DOS_SEQ.Device.AVJ212.EnableCnd := FALSE;
                               VAR_DOS_SEQ.Device.AVJ215.AutoCnd := FALSE;                                             (* STEP: 22 Atmospheric drain valve*)
                               VAR_DOS_SEQ.Device.AVJ215.EnableCnd := FALSE;
                               VAR_DOS_SEQ.Device.AVJ216.AutoCnd := FALSE;                                             (* STEP: 22 Recirculation Valve*)
                               VAR_DOS_SEQ.Device.AVJ216.EnableCnd := FALSE;
                               VAR_DOS_SEQ.Device.AVJ217.AutoCnd := FALSE;                                             (* STEP: 22 Tank Hema Drain Valve*)
                               VAR_DOS_SEQ.Device.AVJ217.EnableCnd := FALSE;
                               VAR_DOS_SEQ.Device.AVJ218.AutoCnd := FALSE;                                             (* STEP: 22 Recirculation Valve*)
                               VAR_DOS_SEQ.Device.AVJ218.EnableCnd := FALSE;
                               VAR_DOS_SEQ.Device.AVJ221.AutoCnd := FALSE;                                             (* STEP: 22 Inlet Loop Valve*)
                               VAR_DOS_SEQ.Device.AVJ221.EnableCnd := FALSE;
                               VAR_DOS_SEQ.Device.AVJ230.AutoCnd := FALSE;                                             (* STEP: 22 *)
                               VAR_DOS_SEQ.Device.AVJ230.EnableCnd := FALSE;
                               VAR_DOS_SEQ.Device.AVJ231.AutoCnd := FALSE;                                             (* STEP: 22 *)
                               VAR_DOS_SEQ.Device.AVJ231.EnableCnd := FALSE;
                               VAR_DOS_SEQ.Device.AVJ232.AutoCnd := FALSE;                                             (* STEP: 22 *)
                               VAR_DOS_SEQ.Device.AVJ232.EnableCnd := FALSE;
                               VAR_DOS_SEQ.Device.AVJ233.AutoCnd := FALSE;                                             (* STEP: 22 *)
                               VAR_DOS_SEQ.Device.AVJ233.EnableCnd := FALSE;
                               VAR_DOS_SEQ.Device.AVJ234.AutoCnd := FALSE;                                             (* STEP: 22 *)
                               VAR_DOS_SEQ.Device.AVJ234.EnableCnd := FALSE;
                               VAR_DOS_SEQ.Device.AVJ235.AutoCnd := FALSE;                                             (* STEP: 22 *)
                               VAR_DOS_SEQ.Device.AVJ235.EnableCnd := FALSE;

                               VAR_DOS_SEQ.Device.LTJ203.ALR_HighLimitEn := TRUE;                                      (* STEP: 22 Hema Tank Level*)
                               VAR_DOS_SEQ.Device.LTJ203.ALR_HighLimitSP := HMI_PAM_3._607;
                               VAR_DOS_SEQ.Device.LTJ203.ALR_LowLimitEn := TRUE;
                               VAR_DOS_SEQ.Device.LTJ203.ALR_LowLimitSP := HMI_PAM_3._606;
                               VAR_DOS_SEQ.Device.LTJ203.SP := HMI_PAM_3._608;
                               VAR_DOS_SEQ.Device.LTJ203.CMP := 2;
                               VAR_DOS_SEQ.Device.LTJ203.MinDev := 0;
                               VAR_DOS_SEQ.Device.LTJ203.MaxDev := 0;

                               VAR_DOS_SEQ.Device.TTJ203.ALR_HighLimitEn := FALSE;                                     (* STEP: 22 Hema Tank Temperature*)
                               VAR_DOS_SEQ.Device.TTJ203.ALR_HighLimitSP := 0;
                               VAR_DOS_SEQ.Device.TTJ203.ALR_LowLimitEn := FALSE;
                               VAR_DOS_SEQ.Device.TTJ203.ALR_LowLimitSP := 0;
                               VAR_DOS_SEQ.Device.TTJ203.SP := HMI_PAM_3._600;
                               VAR_DOS_SEQ.Device.TTJ203.CMP := 0;
                               VAR_DOS_SEQ.Device.TTJ203.MinDev := 0;
                               VAR_DOS_SEQ.Device.TTJ203.MaxDev := 0;

                               VAR_DOS_SEQ.Device.LSJ200.ALR := FALSE;                                                 (* STEP: 22 *)
                               VAR_DOS_SEQ.Device.LSJ200.WAIT_OFF := FALSE;
                               VAR_DOS_SEQ.Device.LSJ200.WAIT_ON := FALSE;

                               VAR_DOS_SEQ.Device.LSJ201.ALR := FALSE;                                                 (* STEP: 22 *)
                               VAR_DOS_SEQ.Device.LSJ201.WAIT_OFF := FALSE;
                               VAR_DOS_SEQ.Device.LSJ201.WAIT_ON := FALSE;

                               VAR_DOS_SEQ.Device.LSJ202.ALR := FALSE;                                                 (* STEP: 22 *)
                               VAR_DOS_SEQ.Device.LSJ202.WAIT_OFF := FALSE;
                               VAR_DOS_SEQ.Device.LSJ202.WAIT_ON := FALSE;

                               VAR_DOS_SEQ.Device.FSJ201.ALR := FALSE;                                                 (* STEP: 22 *)
                               VAR_DOS_SEQ.Device.FSJ201.WAIT_OFF := FALSE;
                               VAR_DOS_SEQ.Device.FSJ201.WAIT_ON := FALSE;

                               VAR_DOS_SEQ.Device.FSJ202.ALR := FALSE;                                                 (* STEP: 22 *)
                               VAR_DOS_SEQ.Device.FSJ202.WAIT_OFF := FALSE;
                               VAR_DOS_SEQ.Device.FSJ202.WAIT_ON := FALSE;

                               VAR_DOS_SEQ.Mem.PBAbortEnable := TRUE;                                                  (* STEP: 22 PB Abort Sequence Enable*)
                               VAR_DOS_SEQ.Mem.PBStopEnable := TRUE;                                                   (* STEP: 22 PB Stop Sequence Enable*)
                               VAR_DOS_SEQ.Mem.PBStartEnable := FALSE;                                                 (* STEP: 22 PB Start Sequence Enable*)
                               VAR_DOS_SEQ.Mem.ContainersStop := TRUE;                                                 (* STEP: 22 *)
                               VAR_DOS_SEQ.Mem.MachineStart := TRUE;                                                   (* STEP: 22 *)
                               VAR_DOS_SEQ.Mem.MachineStop := FALSE;                                                   (* STEP: 22 *)
                               VAR_DOS_SEQ.Mem.DummyBottles := FALSE;                                                  (* STEP: 22 Dummy Bottle Install*)
                               VAR_DOS_SEQ.Mem.PositioningRequest := FALSE;                                            (* STEP: 22 Request of Cam Positioning at height SP of Sequncer*)
                               VAR_DOS_SEQ.Mem.COP_Cycle := FALSE;                                                     (* STEP: 22 COP Cycle Check Requested*)
                               VAR_DOS_SEQ.Mem.LapsCounter := FALSE;                                                   (* STEP: 22 *)
                               VAR_DOS_SEQ.Mem.ValveOpening := FALSE;                                                  (* STEP: 22 *)
                               VAR_DOS_SEQ.Mem.CopAfterCipRequest := FALSE;                                            (* STEP: 22 Request Of Cop After Cip*)

                               VAR_DOS_SEQ.ITC.CIP_CleaningRequest := FALSE;                                           (* STEP: 22 To CIP -> Request of Solution Sending*)
                               VAR_DOS_SEQ.ITC.CIP_Alarm := FALSE;                                                     (* STEP: 22 To CIP -> Critical Alarm Present*)
                               VAR_DOS_SEQ.ITC.CIP_RinseEnded := FALSE;                                                (* STEP: 22 To CIP -> Rinse Finished*)
                               VAR_DOS_SEQ.ITC.CIP_ChangeEnded := FALSE;                                               (* STEP: 22 To CIP -> Change Finished*)
                               VAR_DOS_SEQ.ITC.CIP_DrainRunning := FALSE;                                              (* STEP: 22 To CIP -> Drain Cycle Running*)
                               VAR_DOS_SEQ.ITC.CIP_RinseRunning := FALSE;                                              (* STEP: 22 To CIP -> Rinse Cycle Running*)
                               VAR_DOS_SEQ.ITC.CIP_CleaningRunning := FALSE;                                           (* STEP: 22 To CIP -> Cleaning Cycle Running*)
                               VAR_DOS_SEQ.ITC.CIP_DrainEnded := FALSE;                                                (* STEP: 22 To CIP -> Drain Finished*)
                               VAR_DOS_SEQ.ITC.CIP_FloodingEnded := FALSE;                                             (* STEP: 22 To CIP -> Flooding Finished*)
                               VAR_DOS_SEQ.ITC.CIP_FlipEnable := FALSE;                                                (* STEP: 22 *)
                               VAR_DOS_SEQ.ITC.CIP_CycleEnded := FALSE;                                                (* STEP: 22 *)

                               VAR_DOS_SEQ.ITC.PROD_ReadyForHeating := FALSE;                                          (* STEP: 22 To PASTO -> Filler Ready for Production (Heating)*)
                               VAR_DOS_SEQ.ITC.PROD_DoserInTemperature := FALSE;                                       (* STEP: 22 To PASTO -> Filler Temperature OK (After Heating)*)
                               VAR_DOS_SEQ.ITC.PROD_ProductRequest := TRUE;                                            (* STEP: 22 To PASTO -> Product Request*)
                               VAR_DOS_SEQ.ITC.PROD_DoserOnFillingMode := FALSE;                                       (* STEP: 22 To PASTO -> Product Consumend -Filling Valve Opening*)
                               VAR_DOS_SEQ.ITC.PROD_EndProductionCompleted := FALSE;                                   (* STEP: 22 To PASTO -> End Production Done*)
                               VAR_DOS_SEQ.ITC.PROD_ProductRecoveryEnd := FALSE;                                       (* STEP: 22 To PASTO -> Product Recovery End*)
                               VAR_DOS_SEQ.ITC.PROD_WaterRequestAfterProd := FALSE;                                    (* STEP: 22 To PASTO -> Water Request For Filler Rinse Afetr Production*)

                       23: (* START-UP PRODUCTION -Filling Valve Priming, Filling Valves Opening *)

                               VAR_DOS_SEQ.Device.PPJ201_PID.PID_Enable := FALSE;                                      (* STEP: 23 Doser Recovery Pump*)
                               VAR_DOS_SEQ.Device.PPJ201_PID.PID_Mode := FALSE;
                               VAR_DOS_SEQ.Device.PPJ201_PID.Auto_SP_Value := 0;
                               VAR_DOS_SEQ.Device.PPJ201_PID.FIX_Value := 0;

                               VAR_DOS_SEQ.Device.PPJ202_PID.PID_Enable := FALSE;                                      (* STEP: 23 Doser Recovery Pump*)
                               VAR_DOS_SEQ.Device.PPJ202_PID.PID_Mode := FALSE;
                               VAR_DOS_SEQ.Device.PPJ202_PID.Auto_SP_Value := 0;
                               VAR_DOS_SEQ.Device.PPJ202_PID.FIX_Value := 0;

                               VAR_DOS_SEQ.Device.PPJ203_PID.PID_Enable := FALSE;                                      (* STEP: 23 Diaphragm Pump for Recovery pulp*)
                               VAR_DOS_SEQ.Device.PPJ203_PID.PID_Mode := FALSE;
                               VAR_DOS_SEQ.Device.PPJ203_PID.Auto_SP_Value := 0;
                               VAR_DOS_SEQ.Device.PPJ203_PID.FIX_Value := 0;

                               VAR_DOS_SEQ.Device.MMJ201_PID.PID_Enable := FALSE;                                      (* STEP: 23 Shaker Motor*)
                               VAR_DOS_SEQ.Device.MMJ201_PID.PID_Mode := FALSE;
                               VAR_DOS_SEQ.Device.MMJ201_PID.Auto_SP_Value := 10;
                               VAR_DOS_SEQ.Device.MMJ201_PID.FIX_Value := 0;

                               VAR_DOS_SEQ.Device.RVJ201_PID.PID_Enable := FALSE;                                      (* STEP: 23 *)
                               VAR_DOS_SEQ.Device.RVJ201_PID.PID_Mode := FALSE;
                               VAR_DOS_SEQ.Device.RVJ201_PID.Auto_SP_Value := 0;
                               VAR_DOS_SEQ.Device.RVJ201_PID.FIX_Value := 0;

                               VAR_DOS_SEQ.Device.AVJ201.AutoCnd := TRUE;                                              (* STEP: 23 Inlet Valve*)
                               VAR_DOS_SEQ.Device.AVJ201.EnableCnd := TRUE;
                               VAR_DOS_SEQ.Device.AVJ210.AutoCnd := FALSE;                                             (* STEP: 23 Washing Duct Valve*)
                               VAR_DOS_SEQ.Device.AVJ210.EnableCnd := FALSE;
                               VAR_DOS_SEQ.Device.AVJ211.AutoCnd := FALSE;                                             (* STEP: 23 Sprayball Valve*)
                               VAR_DOS_SEQ.Device.AVJ211.EnableCnd := FALSE;
                               VAR_DOS_SEQ.Device.AVJ212.AutoCnd := FALSE;                                             (* STEP: 23 *)
                               VAR_DOS_SEQ.Device.AVJ212.EnableCnd := FALSE;
                               VAR_DOS_SEQ.Device.AVJ215.AutoCnd := FALSE;                                             (* STEP: 23 Atmospheric drain valve*)
                               VAR_DOS_SEQ.Device.AVJ215.EnableCnd := FALSE;
                               VAR_DOS_SEQ.Device.AVJ216.AutoCnd := FALSE;                                             (* STEP: 23 Recirculation Valve*)
                               VAR_DOS_SEQ.Device.AVJ216.EnableCnd := FALSE;
                               VAR_DOS_SEQ.Device.AVJ217.AutoCnd := FALSE;                                             (* STEP: 23 Tank Hema Drain Valve*)
                               VAR_DOS_SEQ.Device.AVJ217.EnableCnd := FALSE;
                               VAR_DOS_SEQ.Device.AVJ218.AutoCnd := FALSE;                                             (* STEP: 23 Recirculation Valve*)
                               VAR_DOS_SEQ.Device.AVJ218.EnableCnd := FALSE;
                               VAR_DOS_SEQ.Device.AVJ221.AutoCnd := FALSE;                                             (* STEP: 23 Inlet Loop Valve*)
                               VAR_DOS_SEQ.Device.AVJ221.EnableCnd := FALSE;
                               VAR_DOS_SEQ.Device.AVJ230.AutoCnd := FALSE;                                             (* STEP: 23 *)
                               VAR_DOS_SEQ.Device.AVJ230.EnableCnd := FALSE;
                               VAR_DOS_SEQ.Device.AVJ231.AutoCnd := FALSE;                                             (* STEP: 23 *)
                               VAR_DOS_SEQ.Device.AVJ231.EnableCnd := FALSE;
                               VAR_DOS_SEQ.Device.AVJ232.AutoCnd := TRUE;                                              (* STEP: 23 *)
                               VAR_DOS_SEQ.Device.AVJ232.EnableCnd := FALSE;
                               VAR_DOS_SEQ.Device.AVJ233.AutoCnd := FALSE;                                             (* STEP: 23 *)
                               VAR_DOS_SEQ.Device.AVJ233.EnableCnd := FALSE;
                               VAR_DOS_SEQ.Device.AVJ234.AutoCnd := FALSE;                                             (* STEP: 23 *)
                               VAR_DOS_SEQ.Device.AVJ234.EnableCnd := FALSE;
                               VAR_DOS_SEQ.Device.AVJ235.AutoCnd := FALSE;                                             (* STEP: 23 *)
                               VAR_DOS_SEQ.Device.AVJ235.EnableCnd := FALSE;

                               VAR_DOS_SEQ.Device.LTJ203.ALR_HighLimitEn := FALSE;                                     (* STEP: 23 Hema Tank Level*)
                               VAR_DOS_SEQ.Device.LTJ203.ALR_HighLimitSP := 0;
                               VAR_DOS_SEQ.Device.LTJ203.ALR_LowLimitEn := FALSE;
                               VAR_DOS_SEQ.Device.LTJ203.ALR_LowLimitSP := 0;
                               VAR_DOS_SEQ.Device.LTJ203.SP := HMI_PAM_3._608;
                               VAR_DOS_SEQ.Device.LTJ203.CMP := 3;
                               VAR_DOS_SEQ.Device.LTJ203.MinDev := 0;
                               VAR_DOS_SEQ.Device.LTJ203.MaxDev := 0;

                               VAR_DOS_SEQ.Device.TTJ203.ALR_HighLimitEn := FALSE;                                     (* STEP: 23 Hema Tank Temperature*)
                               VAR_DOS_SEQ.Device.TTJ203.ALR_HighLimitSP := 0;
                               VAR_DOS_SEQ.Device.TTJ203.ALR_LowLimitEn := FALSE;
                               VAR_DOS_SEQ.Device.TTJ203.ALR_LowLimitSP := 0;
                               VAR_DOS_SEQ.Device.TTJ203.SP := 0;
                               VAR_DOS_SEQ.Device.TTJ203.CMP := 0;
                               VAR_DOS_SEQ.Device.TTJ203.MinDev := 0;
                               VAR_DOS_SEQ.Device.TTJ203.MaxDev := 0;

                               VAR_DOS_SEQ.Device.LSJ200.ALR := FALSE;                                                 (* STEP: 23 *)
                               VAR_DOS_SEQ.Device.LSJ200.WAIT_OFF := FALSE;
                               VAR_DOS_SEQ.Device.LSJ200.WAIT_ON := FALSE;

                               VAR_DOS_SEQ.Device.LSJ201.ALR := FALSE;                                                 (* STEP: 23 *)
                               VAR_DOS_SEQ.Device.LSJ201.WAIT_OFF := FALSE;
                               VAR_DOS_SEQ.Device.LSJ201.WAIT_ON := FALSE;

                               VAR_DOS_SEQ.Device.LSJ202.ALR := FALSE;                                                 (* STEP: 23 *)
                               VAR_DOS_SEQ.Device.LSJ202.WAIT_OFF := FALSE;
                               VAR_DOS_SEQ.Device.LSJ202.WAIT_ON := TRUE;

                               VAR_DOS_SEQ.Device.FSJ201.ALR := FALSE;                                                 (* STEP: 23 *)
                               VAR_DOS_SEQ.Device.FSJ201.WAIT_OFF := FALSE;
                               VAR_DOS_SEQ.Device.FSJ201.WAIT_ON := FALSE;

                               VAR_DOS_SEQ.Device.FSJ202.ALR := FALSE;                                                 (* STEP: 23 *)
                               VAR_DOS_SEQ.Device.FSJ202.WAIT_OFF := FALSE;
                               VAR_DOS_SEQ.Device.FSJ202.WAIT_ON := FALSE;

                               VAR_DOS_SEQ.Mem.PBAbortEnable := FALSE;                                                 (* STEP: 23 PB Abort Sequence Enable*)
                               VAR_DOS_SEQ.Mem.PBStopEnable := FALSE;                                                  (* STEP: 23 PB Stop Sequence Enable*)
                               VAR_DOS_SEQ.Mem.PBStartEnable := FALSE;                                                 (* STEP: 23 PB Start Sequence Enable*)
                               VAR_DOS_SEQ.Mem.ContainersStop := TRUE;                                                (* STEP: 23 *)
                               VAR_DOS_SEQ.Mem.MachineStart := TRUE;                                                   (* STEP: 23 *)
                               VAR_DOS_SEQ.Mem.MachineStop := FALSE;                                                   (* STEP: 23 *)
                               VAR_DOS_SEQ.Mem.DummyBottles := FALSE;                                                  (* STEP: 23 Dummy Bottle Install*)
                               VAR_DOS_SEQ.Mem.PositioningRequest := FALSE;                                            (* STEP: 23 Request of Cam Positioning at height SP of Sequncer*)
                               VAR_DOS_SEQ.Mem.COP_Cycle := FALSE;                                                     (* STEP: 23 COP Cycle Check Requested*)
                               VAR_DOS_SEQ.Mem.LapsCounter := FALSE;                                                   (* STEP: 23 *)
                               VAR_DOS_SEQ.Mem.ValveOpening := TRUE;                                                   (* STEP: 23 *)
                               VAR_DOS_SEQ.Mem.CopAfterCipRequest := FALSE;                                            (* STEP: 23 Request Of Cop After Cip*)

                               VAR_DOS_SEQ.ITC.CIP_CleaningRequest := FALSE;                                           (* STEP: 23 To CIP -> Request of Solution Sending*)
                               VAR_DOS_SEQ.ITC.CIP_Alarm := FALSE;                                                     (* STEP: 23 To CIP -> Critical Alarm Present*)
                               VAR_DOS_SEQ.ITC.CIP_RinseEnded := FALSE;                                                (* STEP: 23 To CIP -> Rinse Finished*)
                               VAR_DOS_SEQ.ITC.CIP_ChangeEnded := FALSE;                                               (* STEP: 23 To CIP -> Change Finished*)
                               VAR_DOS_SEQ.ITC.CIP_DrainRunning := FALSE;                                              (* STEP: 23 To CIP -> Drain Cycle Running*)
                               VAR_DOS_SEQ.ITC.CIP_RinseRunning := FALSE;                                              (* STEP: 23 To CIP -> Rinse Cycle Running*)
                               VAR_DOS_SEQ.ITC.CIP_CleaningRunning := FALSE;                                           (* STEP: 23 To CIP -> Cleaning Cycle Running*)
                               VAR_DOS_SEQ.ITC.CIP_DrainEnded := FALSE;                                                (* STEP: 23 To CIP -> Drain Finished*)
                               VAR_DOS_SEQ.ITC.CIP_FloodingEnded := FALSE;                                             (* STEP: 23 To CIP -> Flooding Finished*)
                               VAR_DOS_SEQ.ITC.CIP_FlipEnable := FALSE;                                                (* STEP: 23 *)
                               VAR_DOS_SEQ.ITC.CIP_CycleEnded := FALSE;                                                (* STEP: 23 *)

                               VAR_DOS_SEQ.ITC.PROD_ReadyForHeating := FALSE;                                          (* STEP: 23 To PASTO -> Filler Ready for Production (Heating)*)
                               VAR_DOS_SEQ.ITC.PROD_DoserInTemperature := FALSE;                                       (* STEP: 23 To PASTO -> Filler Temperature OK (After Heating)*)
                               VAR_DOS_SEQ.ITC.PROD_ProductRequest := TRUE;                                            (* STEP: 23 To PASTO -> Product Request*)
                               VAR_DOS_SEQ.ITC.PROD_DoserOnFillingMode := FALSE;                                       (* STEP: 23 To PASTO -> Product Consumend -Filling Valve Opening*)
                               VAR_DOS_SEQ.ITC.PROD_EndProductionCompleted := FALSE;                                   (* STEP: 23 To PASTO -> End Production Done*)
                               VAR_DOS_SEQ.ITC.PROD_ProductRecoveryEnd := FALSE;                                       (* STEP: 23 To PASTO -> Product Recovery End*)
                               VAR_DOS_SEQ.ITC.PROD_WaterRequestAfterProd := FALSE;                                    (* STEP: 23 To PASTO -> Water Request For Filler Rinse Afetr Production*)

                       24: (* START-UP PRODUCTION -Filling Valve Priming, Drain Tray Washing *)

                               VAR_DOS_SEQ.Device.PPJ201_PID.PID_Enable := FALSE;                                      (* STEP: 24 Doser Recovery Pump*)
                               VAR_DOS_SEQ.Device.PPJ201_PID.PID_Mode := FALSE;
                               VAR_DOS_SEQ.Device.PPJ201_PID.Auto_SP_Value := 0;
                               VAR_DOS_SEQ.Device.PPJ201_PID.FIX_Value := 0;

                               VAR_DOS_SEQ.Device.PPJ202_PID.PID_Enable := FALSE;                                      (* STEP: 24 Doser Recovery Pump*)
                               VAR_DOS_SEQ.Device.PPJ202_PID.PID_Mode := FALSE;
                               VAR_DOS_SEQ.Device.PPJ202_PID.Auto_SP_Value := 0;
                               VAR_DOS_SEQ.Device.PPJ202_PID.FIX_Value := 0;

                               VAR_DOS_SEQ.Device.PPJ203_PID.PID_Enable := FALSE;                                      (* STEP: 24 Diaphragm Pump for Recovery pulp*)
                               VAR_DOS_SEQ.Device.PPJ203_PID.PID_Mode := FALSE;
                               VAR_DOS_SEQ.Device.PPJ203_PID.Auto_SP_Value := 0;
                               VAR_DOS_SEQ.Device.PPJ203_PID.FIX_Value := 0;

                               VAR_DOS_SEQ.Device.MMJ201_PID.PID_Enable := FALSE;                                      (* STEP: 24 Shaker Motor*)
                               VAR_DOS_SEQ.Device.MMJ201_PID.PID_Mode := FALSE;
                               VAR_DOS_SEQ.Device.MMJ201_PID.Auto_SP_Value := 0;
                               VAR_DOS_SEQ.Device.MMJ201_PID.FIX_Value := 0;

                               VAR_DOS_SEQ.Device.RVJ201_PID.PID_Enable := FALSE;                                      (* STEP: 24 *)
                               VAR_DOS_SEQ.Device.RVJ201_PID.PID_Mode := FALSE;
                               VAR_DOS_SEQ.Device.RVJ201_PID.Auto_SP_Value := 0;
                               VAR_DOS_SEQ.Device.RVJ201_PID.FIX_Value := 0;

                               VAR_DOS_SEQ.Device.AVJ201.AutoCnd := FALSE;                                             (* STEP: 24 Inlet Valve*)
                               VAR_DOS_SEQ.Device.AVJ201.EnableCnd := FALSE;
                               VAR_DOS_SEQ.Device.AVJ210.AutoCnd := TRUE;                                              (* STEP: 24 Washing Duct Valve*)
                               VAR_DOS_SEQ.Device.AVJ210.EnableCnd := FALSE;
                               VAR_DOS_SEQ.Device.AVJ211.AutoCnd := FALSE;                                             (* STEP: 24 Sprayball Valve*)
                               VAR_DOS_SEQ.Device.AVJ211.EnableCnd := FALSE;
                               VAR_DOS_SEQ.Device.AVJ212.AutoCnd := FALSE;                                             (* STEP: 24 *)
                               VAR_DOS_SEQ.Device.AVJ212.EnableCnd := FALSE;
                               VAR_DOS_SEQ.Device.AVJ215.AutoCnd := FALSE;                                             (* STEP: 24 Atmospheric drain valve*)
                               VAR_DOS_SEQ.Device.AVJ215.EnableCnd := FALSE;
                               VAR_DOS_SEQ.Device.AVJ216.AutoCnd := FALSE;                                             (* STEP: 24 Recirculation Valve*)
                               VAR_DOS_SEQ.Device.AVJ216.EnableCnd := FALSE;
                               VAR_DOS_SEQ.Device.AVJ217.AutoCnd := FALSE;                                             (* STEP: 24 Tank Hema Drain Valve*)
                               VAR_DOS_SEQ.Device.AVJ217.EnableCnd := FALSE;
                               VAR_DOS_SEQ.Device.AVJ218.AutoCnd := FALSE;                                             (* STEP: 24 Recirculation Valve*)
                               VAR_DOS_SEQ.Device.AVJ218.EnableCnd := FALSE;
                               VAR_DOS_SEQ.Device.AVJ221.AutoCnd := FALSE;                                             (* STEP: 24 Inlet Loop Valve*)
                               VAR_DOS_SEQ.Device.AVJ221.EnableCnd := FALSE;
                               VAR_DOS_SEQ.Device.AVJ230.AutoCnd := FALSE;                                             (* STEP: 24 *)
                               VAR_DOS_SEQ.Device.AVJ230.EnableCnd := FALSE;
                               VAR_DOS_SEQ.Device.AVJ231.AutoCnd := FALSE;                                             (* STEP: 24 *)
                               VAR_DOS_SEQ.Device.AVJ231.EnableCnd := FALSE;
                               VAR_DOS_SEQ.Device.AVJ232.AutoCnd := FALSE;                                             (* STEP: 24 *)
                               VAR_DOS_SEQ.Device.AVJ232.EnableCnd := FALSE;
                               VAR_DOS_SEQ.Device.AVJ233.AutoCnd := FALSE;                                             (* STEP: 24 *)
                               VAR_DOS_SEQ.Device.AVJ233.EnableCnd := FALSE;
                               VAR_DOS_SEQ.Device.AVJ234.AutoCnd := FALSE;                                             (* STEP: 24 *)
                               VAR_DOS_SEQ.Device.AVJ234.EnableCnd := FALSE;
                               VAR_DOS_SEQ.Device.AVJ235.AutoCnd := FALSE;                                             (* STEP: 24 *)
                               VAR_DOS_SEQ.Device.AVJ235.EnableCnd := FALSE;

                               VAR_DOS_SEQ.Device.LTJ203.ALR_HighLimitEn := FALSE;                                     (* STEP: 24 Hema Tank Level*)
                               VAR_DOS_SEQ.Device.LTJ203.ALR_HighLimitSP := 0;
                               VAR_DOS_SEQ.Device.LTJ203.ALR_LowLimitEn := FALSE;
                               VAR_DOS_SEQ.Device.LTJ203.ALR_LowLimitSP := 0;
                               VAR_DOS_SEQ.Device.LTJ203.SP := 0;
                               VAR_DOS_SEQ.Device.LTJ203.CMP := 0;
                               VAR_DOS_SEQ.Device.LTJ203.MinDev := 0;
                               VAR_DOS_SEQ.Device.LTJ203.MaxDev := 0;

                               VAR_DOS_SEQ.Device.TTJ203.ALR_HighLimitEn := FALSE;                                     (* STEP: 24 Hema Tank Temperature*)
                               VAR_DOS_SEQ.Device.TTJ203.ALR_HighLimitSP := 0;
                               VAR_DOS_SEQ.Device.TTJ203.ALR_LowLimitEn := FALSE;
                               VAR_DOS_SEQ.Device.TTJ203.ALR_LowLimitSP := 0;
                               VAR_DOS_SEQ.Device.TTJ203.SP := 0;
                               VAR_DOS_SEQ.Device.TTJ203.CMP := 0;
                               VAR_DOS_SEQ.Device.TTJ203.MinDev := 0;
                               VAR_DOS_SEQ.Device.TTJ203.MaxDev := 0;

                               VAR_DOS_SEQ.Device.LSJ200.ALR := FALSE;                                                 (* STEP: 24 *)
                               VAR_DOS_SEQ.Device.LSJ200.WAIT_OFF := FALSE;
                               VAR_DOS_SEQ.Device.LSJ200.WAIT_ON := FALSE;

                               VAR_DOS_SEQ.Device.LSJ201.ALR := FALSE;                                                 (* STEP: 24 *)
                               VAR_DOS_SEQ.Device.LSJ201.WAIT_OFF := FALSE;
                               VAR_DOS_SEQ.Device.LSJ201.WAIT_ON := FALSE;

                               VAR_DOS_SEQ.Device.LSJ202.ALR := FALSE;                                                 (* STEP: 24 *)
                               VAR_DOS_SEQ.Device.LSJ202.WAIT_OFF := FALSE;
                               VAR_DOS_SEQ.Device.LSJ202.WAIT_ON := FALSE;

                               VAR_DOS_SEQ.Device.FSJ201.ALR := FALSE;                                                 (* STEP: 24 *)
                               VAR_DOS_SEQ.Device.FSJ201.WAIT_OFF := FALSE;
                               VAR_DOS_SEQ.Device.FSJ201.WAIT_ON := FALSE;

                               VAR_DOS_SEQ.Device.FSJ202.ALR := FALSE;                                                 (* STEP: 24 *)
                               VAR_DOS_SEQ.Device.FSJ202.WAIT_OFF := FALSE;
                               VAR_DOS_SEQ.Device.FSJ202.WAIT_ON := FALSE;

                               VAR_DOS_SEQ.Mem.PBAbortEnable := FALSE;                                                 (* STEP: 24 PB Abort Sequence Enable*)
                               VAR_DOS_SEQ.Mem.PBStopEnable := FALSE;                                                  (* STEP: 24 PB Stop Sequence Enable*)
                               VAR_DOS_SEQ.Mem.PBStartEnable := FALSE;                                                 (* STEP: 24 PB Start Sequence Enable*)
                               VAR_DOS_SEQ.Mem.ContainersStop := TRUE;                                                (* STEP: 24 *)
                               VAR_DOS_SEQ.Mem.MachineStart := FALSE;                                                  (* STEP: 24 *)
                               VAR_DOS_SEQ.Mem.MachineStop := FALSE;                                                   (* STEP: 24 *)
                               VAR_DOS_SEQ.Mem.DummyBottles := FALSE;                                                  (* STEP: 24 Dummy Bottle Install*)
                               VAR_DOS_SEQ.Mem.PositioningRequest := FALSE;                                            (* STEP: 24 Request of Cam Positioning at height SP of Sequncer*)
                               VAR_DOS_SEQ.Mem.COP_Cycle := FALSE;                                                     (* STEP: 24 COP Cycle Check Requested*)
                               VAR_DOS_SEQ.Mem.LapsCounter := FALSE;                                                   (* STEP: 24 *)
                               VAR_DOS_SEQ.Mem.ValveOpening := FALSE;                                                  (* STEP: 24 *)
                               VAR_DOS_SEQ.Mem.CopAfterCipRequest := FALSE;                                            (* STEP: 24 Request Of Cop After Cip*)

                               VAR_DOS_SEQ.ITC.CIP_CleaningRequest := FALSE;                                           (* STEP: 24 To CIP -> Request of Solution Sending*)
                               VAR_DOS_SEQ.ITC.CIP_Alarm := FALSE;                                                     (* STEP: 24 To CIP -> Critical Alarm Present*)
                               VAR_DOS_SEQ.ITC.CIP_RinseEnded := FALSE;                                                (* STEP: 24 To CIP -> Rinse Finished*)
                               VAR_DOS_SEQ.ITC.CIP_ChangeEnded := FALSE;                                               (* STEP: 24 To CIP -> Change Finished*)
                               VAR_DOS_SEQ.ITC.CIP_DrainRunning := FALSE;                                              (* STEP: 24 To CIP -> Drain Cycle Running*)
                               VAR_DOS_SEQ.ITC.CIP_RinseRunning := FALSE;                                              (* STEP: 24 To CIP -> Rinse Cycle Running*)
                               VAR_DOS_SEQ.ITC.CIP_CleaningRunning := FALSE;                                           (* STEP: 24 To CIP -> Cleaning Cycle Running*)
                               VAR_DOS_SEQ.ITC.CIP_DrainEnded := FALSE;                                                (* STEP: 24 To CIP -> Drain Finished*)
                               VAR_DOS_SEQ.ITC.CIP_FloodingEnded := FALSE;                                             (* STEP: 24 To CIP -> Flooding Finished*)
                               VAR_DOS_SEQ.ITC.CIP_FlipEnable := FALSE;                                                (* STEP: 24 *)
                               VAR_DOS_SEQ.ITC.CIP_CycleEnded := FALSE;                                                (* STEP: 24 *)

                               VAR_DOS_SEQ.ITC.PROD_ReadyForHeating := FALSE;                                          (* STEP: 24 To PASTO -> Filler Ready for Production (Heating)*)
                               VAR_DOS_SEQ.ITC.PROD_DoserInTemperature := FALSE;                                       (* STEP: 24 To PASTO -> Filler Temperature OK (After Heating)*)
                               VAR_DOS_SEQ.ITC.PROD_ProductRequest := TRUE;                                            (* STEP: 24 To PASTO -> Product Request*)
                               VAR_DOS_SEQ.ITC.PROD_DoserOnFillingMode := FALSE;                                       (* STEP: 24 To PASTO -> Product Consumend -Filling Valve Opening*)
                               VAR_DOS_SEQ.ITC.PROD_EndProductionCompleted := FALSE;                                   (* STEP: 24 To PASTO -> End Production Done*)
                               VAR_DOS_SEQ.ITC.PROD_ProductRecoveryEnd := FALSE;                                       (* STEP: 24 To PASTO -> Product Recovery End*)
                               VAR_DOS_SEQ.ITC.PROD_WaterRequestAfterProd := FALSE;                                    (* STEP: 24 To PASTO -> Water Request For Filler Rinse Afetr Production*)

                       25..29: (* Spare Steps *)

                       30: (* START-UP PRODUCTION -Wait For Product Tank at Set-Point Level *)

                               VAR_DOS_SEQ.Device.PPJ201_PID.PID_Enable := FALSE;                                      (* STEP: 30 Doser Recovery Pump*)
                               VAR_DOS_SEQ.Device.PPJ201_PID.PID_Mode := FALSE;
                               VAR_DOS_SEQ.Device.PPJ201_PID.Auto_SP_Value := 0;
                               VAR_DOS_SEQ.Device.PPJ201_PID.FIX_Value := 0;

                               VAR_DOS_SEQ.Device.PPJ202_PID.PID_Enable := FALSE;                                      (* STEP: 30 Doser Recovery Pump*)
                               VAR_DOS_SEQ.Device.PPJ202_PID.PID_Mode := FALSE;
                               VAR_DOS_SEQ.Device.PPJ202_PID.Auto_SP_Value := 0;
                               VAR_DOS_SEQ.Device.PPJ202_PID.FIX_Value := 0;

                               VAR_DOS_SEQ.Device.PPJ203_PID.PID_Enable := FALSE;                                      (* STEP: 30 Diaphragm Pump for Recovery pulp*)
                               VAR_DOS_SEQ.Device.PPJ203_PID.PID_Mode := FALSE;
                               VAR_DOS_SEQ.Device.PPJ203_PID.Auto_SP_Value := 0;
                               VAR_DOS_SEQ.Device.PPJ203_PID.FIX_Value := 0;

                               VAR_DOS_SEQ.Device.MMJ201_PID.PID_Enable := TRUE;                                       (* STEP: 30 Shaker Motor*)
                               VAR_DOS_SEQ.Device.MMJ201_PID.PID_Mode := TRUE;
                               VAR_DOS_SEQ.Device.MMJ201_PID.Auto_SP_Value := 20;
                               VAR_DOS_SEQ.Device.MMJ201_PID.FIX_Value := 0;

                               VAR_DOS_SEQ.Device.RVJ201_PID.PID_Enable := FALSE;                                      (* STEP: 30 *)
                               VAR_DOS_SEQ.Device.RVJ201_PID.PID_Mode := FALSE;
                               VAR_DOS_SEQ.Device.RVJ201_PID.Auto_SP_Value := 0;
                               VAR_DOS_SEQ.Device.RVJ201_PID.FIX_Value := 0;

                               VAR_DOS_SEQ.Device.AVJ201.AutoCnd := TRUE;                                              (* STEP: 30 Inlet Valve*)
                               VAR_DOS_SEQ.Device.AVJ201.EnableCnd := TRUE;
                               VAR_DOS_SEQ.Device.AVJ210.AutoCnd := FALSE;                                             (* STEP: 30 Washing Duct Valve*)
                               VAR_DOS_SEQ.Device.AVJ210.EnableCnd := FALSE;
                               VAR_DOS_SEQ.Device.AVJ211.AutoCnd := FALSE;                                             (* STEP: 30 Sprayball Valve*)
                               VAR_DOS_SEQ.Device.AVJ211.EnableCnd := FALSE;
                               VAR_DOS_SEQ.Device.AVJ212.AutoCnd := FALSE;                                             (* STEP: 30 *)
                               VAR_DOS_SEQ.Device.AVJ212.EnableCnd := FALSE;
                               VAR_DOS_SEQ.Device.AVJ215.AutoCnd := FALSE;                                             (* STEP: 30 Atmospheric drain valve*)
                               VAR_DOS_SEQ.Device.AVJ215.EnableCnd := FALSE;
                               VAR_DOS_SEQ.Device.AVJ216.AutoCnd := FALSE;                                             (* STEP: 30 Recirculation Valve*)
                               VAR_DOS_SEQ.Device.AVJ216.EnableCnd := FALSE;
                               VAR_DOS_SEQ.Device.AVJ217.AutoCnd := FALSE;                                             (* STEP: 30 Tank Hema Drain Valve*)
                               VAR_DOS_SEQ.Device.AVJ217.EnableCnd := FALSE;
                               VAR_DOS_SEQ.Device.AVJ218.AutoCnd := FALSE;                                             (* STEP: 30 Recirculation Valve*)
                               VAR_DOS_SEQ.Device.AVJ218.EnableCnd := FALSE;
                               VAR_DOS_SEQ.Device.AVJ221.AutoCnd := FALSE;                                             (* STEP: 30 Inlet Loop Valve*)
                               VAR_DOS_SEQ.Device.AVJ221.EnableCnd := FALSE;
                               VAR_DOS_SEQ.Device.AVJ230.AutoCnd := FALSE;                                             (* STEP: 30 *)
                               VAR_DOS_SEQ.Device.AVJ230.EnableCnd := FALSE;
                               VAR_DOS_SEQ.Device.AVJ231.AutoCnd := FALSE;                                             (* STEP: 30 *)
                               VAR_DOS_SEQ.Device.AVJ231.EnableCnd := FALSE;
                               VAR_DOS_SEQ.Device.AVJ232.AutoCnd := FALSE;                                             (* STEP: 30 *)
                               VAR_DOS_SEQ.Device.AVJ232.EnableCnd := FALSE;
                               VAR_DOS_SEQ.Device.AVJ233.AutoCnd := FALSE;                                             (* STEP: 30 *)
                               VAR_DOS_SEQ.Device.AVJ233.EnableCnd := FALSE;
                               VAR_DOS_SEQ.Device.AVJ234.AutoCnd := FALSE;                                             (* STEP: 30 *)
                               VAR_DOS_SEQ.Device.AVJ234.EnableCnd := FALSE;
                               VAR_DOS_SEQ.Device.AVJ235.AutoCnd := FALSE;                                             (* STEP: 30 *)
                               VAR_DOS_SEQ.Device.AVJ235.EnableCnd := FALSE;

                               VAR_DOS_SEQ.Device.LTJ203.ALR_HighLimitEn := TRUE;                                      (* STEP: 30 Hema Tank Level*)
                               VAR_DOS_SEQ.Device.LTJ203.ALR_HighLimitSP := HMI_PAM_3._607;
                               VAR_DOS_SEQ.Device.LTJ203.ALR_LowLimitEn := FALSE;
                               VAR_DOS_SEQ.Device.LTJ203.ALR_LowLimitSP := 0;
                               VAR_DOS_SEQ.Device.LTJ203.SP := HMI_PAM_3._608;
                               VAR_DOS_SEQ.Device.LTJ203.CMP := 2;
                               VAR_DOS_SEQ.Device.LTJ203.MinDev := 0;
                               VAR_DOS_SEQ.Device.LTJ203.MaxDev := 0;

                               VAR_DOS_SEQ.Device.TTJ203.ALR_HighLimitEn := TRUE;                                      (* STEP: 30 Hema Tank Temperature*)
                               VAR_DOS_SEQ.Device.TTJ203.ALR_HighLimitSP := HMI_PAM_3._604;
                               VAR_DOS_SEQ.Device.TTJ203.ALR_LowLimitEn := TRUE;
                               VAR_DOS_SEQ.Device.TTJ203.ALR_LowLimitSP := HMI_PAM_3._603;
                               VAR_DOS_SEQ.Device.TTJ203.SP := HMI_PAM_3._600;
                               VAR_DOS_SEQ.Device.TTJ203.CMP := 2;
                               VAR_DOS_SEQ.Device.TTJ203.MinDev := 0;
                               VAR_DOS_SEQ.Device.TTJ203.MaxDev := 0;

                               VAR_DOS_SEQ.Device.LSJ200.ALR := FALSE;                                                 (* STEP: 30 *)
                               VAR_DOS_SEQ.Device.LSJ200.WAIT_OFF := FALSE;
                               VAR_DOS_SEQ.Device.LSJ200.WAIT_ON := FALSE;

                               VAR_DOS_SEQ.Device.LSJ201.ALR := FALSE;                                                 (* STEP: 30 *)
                               VAR_DOS_SEQ.Device.LSJ201.WAIT_OFF := FALSE;
                               VAR_DOS_SEQ.Device.LSJ201.WAIT_ON := FALSE;

                               VAR_DOS_SEQ.Device.LSJ202.ALR := FALSE;                                                 (* STEP: 30 *)
                               VAR_DOS_SEQ.Device.LSJ202.WAIT_OFF := FALSE;
                               VAR_DOS_SEQ.Device.LSJ202.WAIT_ON := FALSE;

                               VAR_DOS_SEQ.Device.FSJ201.ALR := FALSE;                                                 (* STEP: 30 *)
                               VAR_DOS_SEQ.Device.FSJ201.WAIT_OFF := FALSE;
                               VAR_DOS_SEQ.Device.FSJ201.WAIT_ON := FALSE;

                               VAR_DOS_SEQ.Device.FSJ202.ALR := FALSE;                                                 (* STEP: 30 *)
                               VAR_DOS_SEQ.Device.FSJ202.WAIT_OFF := FALSE;
                               VAR_DOS_SEQ.Device.FSJ202.WAIT_ON := FALSE;

                               VAR_DOS_SEQ.Mem.PBAbortEnable := TRUE;                                                  (* STEP: 30 PB Abort Sequence Enable*)
                               VAR_DOS_SEQ.Mem.PBStopEnable := TRUE;                                                   (* STEP: 30 PB Stop Sequence Enable*)
                               VAR_DOS_SEQ.Mem.PBStartEnable := FALSE;                                                 (* STEP: 30 PB Start Sequence Enable*)
                               VAR_DOS_SEQ.Mem.ContainersStop := TRUE;                                                (* STEP: 30 *)
                               VAR_DOS_SEQ.Mem.MachineStart := FALSE;                                                  (* STEP: 30 *)
                               VAR_DOS_SEQ.Mem.MachineStop := FALSE;                                                   (* STEP: 30 *)
                               VAR_DOS_SEQ.Mem.DummyBottles := FALSE;                                                  (* STEP: 30 Dummy Bottle Install*)
                               VAR_DOS_SEQ.Mem.PositioningRequest := FALSE;                                            (* STEP: 30 Request of Cam Positioning at height SP of Sequncer*)
                               VAR_DOS_SEQ.Mem.COP_Cycle := FALSE;                                                     (* STEP: 30 COP Cycle Check Requested*)
                               VAR_DOS_SEQ.Mem.LapsCounter := FALSE;                                                   (* STEP: 30 *)
                               VAR_DOS_SEQ.Mem.ValveOpening := FALSE;                                                  (* STEP: 30 *)
                               VAR_DOS_SEQ.Mem.CopAfterCipRequest := FALSE;                                            (* STEP: 30 Request Of Cop After Cip*)
```
